// TIA Portal project "Paletizace trayů" (V14)

(* hardware
DEVICE "ET 200S station_1"  ET 200S station
   slot 0: "Rack_0"  Rail
   slot 2: "PLC_1"  IM 151-8 PN/DP CPU  6ES7 151-8AB01-0AB0  V3.2
      slot 1: "PROFINET interface_1"  PN-IO
         slot 1: "Port_1"  Port
         slot 2: "Port_2"  Port
         slot 3: "Port_3"  Port
   slot 4: "PM-E 24VDC_1"  PM-E 24VDC  6ES7 138-4CA01-0AA0
   slot 5: "4SI IO link_1"  4SI IO link  6ES7 138-4GA50-0AB0
   slot 6: "4SI IO link_2"  4SI IO link  6ES7 138-4GA50-0AB0
   slot 7: "4SI IO link_3"  4SI IO link  6ES7 138-4GA50-0AB0
   slot 8: "4SI IO link_4"  4SI IO link  6ES7 138-4GA50-0AB0
   slot 9: "PM-E 24VDC_2"  PM-E 24VDC  6ES7 138-4CA01-0AA0
   slot 10: "8DI x 24VDC_1"  8DI x 24VDC  6ES7 131-4BF00-0AA0
   slot 11: "8DI x 24VDC_2"  8DI x 24VDC  6ES7 131-4BF00-0AA0
   slot 12: "8DI x 24VDC_3"  8DI x 24VDC  6ES7 131-4BF00-0AA0
   slot 13: "8DI x 24VDC_4"  8DI x 24VDC  6ES7 131-4BF00-0AA0
   slot 14: "8DI x 24VDC_5"  8DI x 24VDC  6ES7 131-4BF00-0AA0
   slot 15: "8DI x 24VDC_6"  8DI x 24VDC  6ES7 131-4BF00-0AA0
   slot 16: "8DI x 24VDC_7"  8DI x 24VDC  6ES7 131-4BF00-0AA0
   slot 17: "8DI x 24VDC_8"  8DI x 24VDC  6ES7 131-4BF00-0AA0
   slot 18: "8DI x 24VDC_9"  8DI x 24VDC  6ES7 131-4BF00-0AA0
   slot 19: "8DI x 24VDC_10"  8DI x 24VDC  6ES7 131-4BF00-0AA0
   slot 20: "8DI x 24VDC_11"  8DI x 24VDC  6ES7 131-4BF00-0AA0
   slot 21: "8DI x 24VDC_12"  8DI x 24VDC  6ES7 131-4BF00-0AA0
   slot 22: "8DI x 24VDC_13"  8DI x 24VDC  6ES7 131-4BF00-0AA0
   slot 23: "8DI x 24VDC_14"  8DI x 24VDC  6ES7 131-4BF00-0AA0
   slot 24: "8DI x 24VDC_15"  8DI x 24VDC  6ES7 131-4BF00-0AA0
   slot 25: "8DI x 24VDC_16"  8DI x 24VDC  6ES7 131-4BF00-0AA0
   slot 26: "PM-E 24VDC_3"  PM-E 24VDC  6ES7 138-4CA01-0AA0
   slot 27: "8DO x 24VDC / 0.5A_1"  8DO x 24VDC / 0.5A  6ES7 132-4BF00-0AA0
   slot 28: "8DO x 24VDC / 0.5A_2"  8DO x 24VDC / 0.5A  6ES7 132-4BF00-0AA0
   slot 29: "PM-E 24VDC_4"  PM-E 24VDC  6ES7 138-4CA01-0AA0
   slot 30: "8DO x 24VDC / 0.5A_3"  8DO x 24VDC / 0.5A  6ES7 132-4BF00-0AA0
   slot 31: "8DO x 24VDC / 0.5A_4"  8DO x 24VDC / 0.5A  6ES7 132-4BF00-0AA0
   slot 32: "8DO x 24VDC / 0.5A_5"  8DO x 24VDC / 0.5A  6ES7 132-4BF00-0AA0
   slot 33: "8DO x 24VDC / 0.5A_6"  8DO x 24VDC / 0.5A  6ES7 132-4BF00-0AA0
   slot 34: "8DO x 24VDC / 0.5A_7"  8DO x 24VDC / 0.5A  6ES7 132-4BF00-0AA0
   slot 35: "8DO x 24VDC / 0.5A_8"  8DO x 24VDC / 0.5A  6ES7 132-4BF00-0AA0
   slot 36: "8DO x 24VDC / 0.5A_9"  8DO x 24VDC / 0.5A  6ES7 132-4BF00-0AA0
   slot 37: "8DO x 24VDC / 0.5A_10"  8DO x 24VDC / 0.5A  6ES7 132-4BF00-0AA0
   slot 38: "8DO x 24VDC / 0.5A_11"  8DO x 24VDC / 0.5A  6ES7 132-4BF00-0AA0
   slot 39: "PM-E 24VDC_5"  PM-E 24VDC  6ES7 138-4CA01-0AA0
   slot 40: "8DO x 24VDC / 0.5A_12"  8DO x 24VDC / 0.5A  6ES7 132-4BF00-0AA0
   slot 41: "8DO x 24VDC / 0.5A_13"  8DO x 24VDC / 0.5A  6ES7 132-4BF00-0AA0
   slot 42: "8DO x 24VDC / 0.5A_14"  8DO x 24VDC / 0.5A  6ES7 132-4BF00-0AA0
   slot 43: "8DO x 24VDC / 0.5A_15"  8DO x 24VDC / 0.5A  6ES7 132-4BF00-0AA0
   slot 44: "8DO x 24VDC / 0.5A_16"  8DO x 24VDC / 0.5A  6ES7 132-4BF00-0AA0
   slot 45: "8DO x 24VDC / 0.5A_17"  8DO x 24VDC / 0.5A  6ES7 132-4BF00-0AA0
   slot 46: "8DO x 24VDC / 0.5A_18"  8DO x 24VDC / 0.5A  6ES7 132-4BF00-0AA0
   slot 47: "8DO x 24VDC / 0.5A_19"  8DO x 24VDC / 0.5A  6ES7 132-4BF00-0AA0
   slot 48: "8DO x 24VDC / 0.5A_20"  8DO x 24VDC / 0.5A  6ES7 132-4BF00-0AA0
*)

// ===== PLC "PLC_1"  IM 151-8 PN/DP CPU =====

TYPE "Artikl2"
   STRUCT
      Cislo : Int;
      Pocet : Int;
      Novy : Bool;
      Mlecny : Bool;
   END_STRUCT;
END_TYPE

TYPE "Artikl"
   STRUCT
      Novy : Bool;
      Mlecny : Bool;
      Mlecny4 : Bool;
      Mlecny6 : Bool;
      Mlecny8 : Bool;
      Mlecny9 : Bool;
      Mlecny99 : Bool;
      Mlecny9999 : Bool;
      Cislo : Word;
      Pocet : Word;
   END_STRUCT;
END_TYPE

DATA_BLOCK "Data"   // DB1
{ S7_Optimized_Access := 'FALSE' }
VERSION : 0.1
   VAR
      Prvni : Bool;
      Druha : Bool;
      Cislo : Int;
      DruheCislo : Int;
   END_VAR
BEGIN
END_DATA_BLOCK

DATA_BLOCK "Data_block_1"   // DB2
{ S7_Optimized_Access := 'FALSE' }
VERSION : 0.1
   VAR
      moje : Struct
         aa : Bool;
         aaaa : Bool;
      END_STRUCT;
      dd : Bool;
   END_VAR
BEGIN
END_DATA_BLOCK

DATA_BLOCK "Data_block_2"   // DB3
{ S7_Optimized_Access := 'FALSE' }
VERSION : 0.1
BEGIN
END_DATA_BLOCK

DATA_BLOCK "DataPole"   // DB4
{ S7_Optimized_Access := 'FALSE' }
VERSION : 0.1
   VAR
      Artikly : Array[0..100] of "Artikl2";
      Konci : Bool;
   END_VAR
BEGIN
END_DATA_BLOCK

DATA_BLOCK "Block_1_DB"   // DB5
{ S7_Optimized_Access := 'FALSE' }
VERSION : 0.1
// stored: InstanceOfName Block_1
"Block_1"
BEGIN
END_DATA_BLOCK

DATA_BLOCK "ArtiklDB"   // DB6
{ S7_Optimized_Access := 'FALSE' }
VERSION : 0.1
   VAR
      Artikl : "Artikl";
   END_VAR
BEGIN
END_DATA_BLOCK

DATA_BLOCK "Data_block_3"   // DB9
{ S7_Optimized_Access := 'FALSE' }
VERSION : 0.1
   VAR
      artikl : Struct
         Novy : Bool;
         Mlecny : Bool;
         Mlecny4 : Bool;
         Mlecny6 : Bool;
         Mlecny8 : Bool;
         Mlecny9 : Bool;
         Mlecny99 : Bool;
         Mlecny9999 : Bool;
         Cislo : Word;
         Pocet : Word;
      END_STRUCT;
   END_VAR
BEGIN
END_DATA_BLOCK

DATA_BLOCK "Artikly"   // DB10
{ S7_Optimized_Access := 'FALSE' }
VERSION : 0.1
   VAR
      Artikly : Array[0..100] of "Artikl";
   END_VAR
BEGIN
END_DATA_BLOCK

FUNCTION_BLOCK "Block_1"   // FB1, LAD
{ S7_Optimized_Access := 'FALSE' }
VERSION : 0.1
BEGIN
END_FUNCTION_BLOCK

ORGANIZATION_BLOCK "Main"   // OB1, LAD
TITLE = "Main Program Sweep (Cycle)"
{ S7_Optimized_Access := 'FALSE' }
VERSION : 0.1
   VAR_TEMP
      OB1_EV_CLASS : Byte;   // Bits 0-3 = 1 (Coming event), Bits 4-7 = 1 (Event class 1)
      OB1_SCAN_1 : Byte;   // 1 (Cold restart scan 1 of OB 1), 3 (Scan 2-n of OB 1)
      OB1_PRIORITY : Byte;   // Priority of OB Execution
      OB1_OB_NUMBR : Byte;   // 1 (Organization block 1, OB1)
      OB1_RESERVED_1 : Byte;   // Reserved for system
      OB1_RESERVED_2 : Byte;   // Reserved for system
      OB1_PREV_CYCLE : Int;   // Cycle time of previous OB1 scan (milliseconds)
      OB1_MIN_CYCLE : Int;   // Minimum cycle time of OB1 (milliseconds)
      OB1_MAX_CYCLE : Int;   // Maximum cycle time of OB1 (milliseconds)
      OB1_DATE_TIME : Date_And_Time;   // Date and time OB1 started
   END_VAR
BEGIN

REGION Network 1
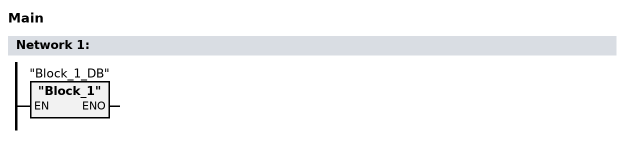
   RUNG wire#powerrail
      "Block_1_DB"()
   END_RUNG
   // the same network as SCL:
   "Block_1_DB"();   // "Block_1"
END_REGION
END_ORGANIZATION_BLOCK